{attribute addProperty BoxType "EJ2522-0000-0022"}
{attribute addProperty Id "StatusAT %I*Status_2BCA7A521620Counter_valueAT %I*UDINT32417"}
{attribute addProperty CRC "3623391603"}
{attribute addProperty SizeInBites "48"}
{attribute addProperty SizeInBytes "6"}
TYPE ENC_Status_Channel_D7F89173 :
STRUCT
	{attribute addProperty Name "Status"}
	Status AT %I* : Status_2BCA7A52;
	{attribute addProperty Name "Counter_value"}
	Counter_value AT %I* : UDINT;
END_STRUCT
END_TYPE

(* stored: Version 1.2.0.0, ProductVersion 3.1.4024.9
   DUT ENC_Status_Channel_D7F89173: Id {8f81ccbc-dcb4-4414-8f36-eac02fb936a6} *)
